// TIA Portal V20 export
DATA_BLOCK "LDrvSafe_SinaTlg701Control_DB_DR10"   // DB370
FAMILY : LDrvSafe
VERSION : 2.0
// stored: InstanceOfName LDrvSafe_SinaTlg701Control, InstanceOfType FB, Namespace Unit1
"LDrvSafe_SinaTlg701Control"
   // VAR_INPUT
   //    enable : Bool := FALSE;
   //    closeBrake : Bool := FALSE;
   //    selectBrakeTest : Bool := FALSE;
   //    startBrakeTest : Bool := FALSE;
   //    brakeSelection : Bool := FALSE;
   //    selectDirectionOfRotation : Bool := FALSE;
   //    selectTestSequence : Bool := FALSE;
   //    statusOfExternalBrake : Bool := FALSE;
   //    hardwareId : HW_IO := 0;
   // END_VAR
   // VAR_OUTPUT
   //    valid { ExternalWritable := 'False'} : Bool := FALSE;
   //    busy { ExternalWritable := 'False'} : Bool := FALSE;
   //    error { ExternalWritable := 'False'} : Bool := FALSE;
   //    status { ExternalWritable := 'False'} : Word := 16#7000;
   // END_VAR
   // VAR
   //    statEnableOld { ExternalVisible := 'False'; ExternalWritable := 'False'} : Bool := FALSE;
   //    statValid { ExternalVisible := 'False'; ExternalWritable := 'False'} : Bool := FALSE;
   //    statBusy { ExternalVisible := 'False'; ExternalWritable := 'False'} : Bool := FALSE;
   //    statError { ExternalVisible := 'False'; ExternalWritable := 'False'} : Bool := FALSE;
   //    statErrorWrite { ExternalVisible := 'False'; ExternalWritable := 'False'} : Bool := FALSE;
   //    statStatus { ExternalVisible := 'False'; ExternalWritable := 'False'} : Word := 16#7000;
   //    statStatusWrite { ExternalVisible := 'False'; ExternalWritable := 'False'} : DWord := 16#0000_0000;
   //    statFBState { ExternalVisible := 'False'; ExternalWritable := 'False'} : DInt := 0;
   //    statDisablingCompleted { ExternalVisible := 'False'; ExternalWritable := 'False'} : Bool := FALSE;
   //    statSendBuf { ExternalVisible := 'False'; ExternalWritable := 'False'} : "LDrvSafe_typeSinaTlg701Control";
   //    instWriteTlg701 { ExternalVisible := 'False'; ExternalWritable := 'False'} : SETIO_PART;
   // END_VAR
BEGIN
   statSendBuf.S_STW1B.reserved8 := FALSE;
   statSendBuf.S_STW1B.reserved9 := FALSE;
   statSendBuf.S_STW1B.reserved10 := FALSE;
   statSendBuf.S_STW1B.reserved11 := FALSE;
   statSendBuf.S_STW1B.reserved12 := FALSE;
   statSendBuf.S_STW1B.closeBrake := FALSE;
   statSendBuf.S_STW1B.reserved14 := FALSE;
   statSendBuf.S_STW1B.reserved15 := FALSE;
   statSendBuf.S_STW1B.reserved0 := FALSE;
   statSendBuf.S_STW1B.reserved1 := FALSE;
   statSendBuf.S_STW1B.reserved2 := FALSE;
   statSendBuf.S_STW1B.reserved3 := FALSE;
   statSendBuf.S_STW1B.reserved4 := FALSE;
   statSendBuf.S_STW1B.reserved5 := FALSE;
   statSendBuf.S_STW1B.reserved6 := FALSE;
   statSendBuf.S_STW1B.reserved7 := FALSE;
   statSendBuf.S_STW3B.reserved2 := FALSE;
   statSendBuf.S_STW3B.reserved3 := FALSE;
   statSendBuf.S_STW3B.reserved4 := FALSE;
   statSendBuf.S_STW3B.reserved5 := FALSE;
   statSendBuf.S_STW3B.reserved6 := FALSE;
   statSendBuf.S_STW3B.reserved7 := FALSE;
   statSendBuf.S_STW3B.reserved8 := FALSE;
   statSendBuf.S_STW3B.reserved9 := FALSE;
   statSendBuf.S_STW3B.selectBrakeTest := FALSE;
   statSendBuf.S_STW3B.startBrakeTest := FALSE;
   statSendBuf.S_STW3B.brakeSelection := FALSE;
   statSendBuf.S_STW3B.selectDirectionOfRotation := FALSE;
   statSendBuf.S_STW3B.selectTestSequence := FALSE;
   statSendBuf.S_STW3B.statusOfExternalBrake := FALSE;
   statSendBuf.S_STW3B.reserved0 := FALSE;
   statSendBuf.S_STW3B.reserved1 := FALSE;
   instWriteTlg701.ID := 0;
   instWriteTlg701.OFFSET := 0;
   instWriteTlg701.LEN := 0;
   instWriteTlg701.STATUS := 16#0000_0000;
   instWriteTlg701.ERROR := FALSE;
END_DATA_BLOCK
